FUNCTION TryConvert_UDINT_TO_TIME : BOOL
VAR_INPUT
	in : UDINT;
	out : REFERENCE TO TIME;
END_VAR

out := UDINT_TO_TIME(in);
TryConvert_UDINT_TO_TIME := TRUE;

END_FUNCTION

(* stored: Version 1.1.0.1, ProductVersion 3.1.4024.12
   POU TryConvert_UDINT_TO_TIME: Id {bd3dbe97-c879-4091-a6ad-a3b6c107db56}, SpecialFunc None *)
